PROGRAM PG_Sonne
VAR
	Sun_history: FB_DataHistory_Int;
	INT_TRIG_0: INT_TRIG;
	FB_Sonne_1: FB_Sonne;
	R_TRIG_0: R_TRIG;
END_VAR
VAR // added by the converter: edge detectors and wires of the graphical bodies
    _w1 : BOOL;
END_VAR

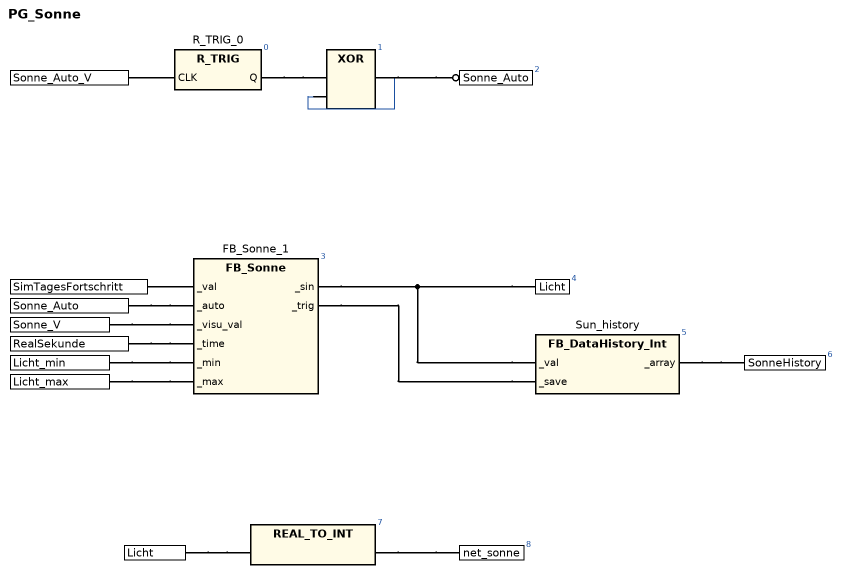
R_TRIG_0(CLK := Sonne_Auto_V); // R_TRIG
_w1 := R_TRIG_0.Q XOR _w1;
Sonne_Auto := NOT _w1;
FB_Sonne_1(
    _val := SimTagesFortschritt,
    _auto := Sonne_Auto,
    _visu_val := Sonne_V,
    _time := RealSekunde,
    _min := Licht_min,
    _max := Licht_max); // FB_Sonne
Licht := FB_Sonne_1._sin;
Sun_history(_val := FB_Sonne_1._sin, _save := FB_Sonne_1._trig); // FB_DataHistory_Int
SonneHistory := Sun_history._array;
net_sonne := REAL_TO_INT(Licht);

END_PROGRAM

(* stored: Version 1.1.0.1, ProductVersion 3.1.4018.5
   POU PG_Sonne: Id {6f2d8c91-1a48-4e18-a6d3-ae78ffda30c8}, SpecialFunc None *)
